FUNCTION Reader : INT
VAR
	numbers : ARRAY[1..5] OF INT := [12, 3, 6, 9];  // Your set of numbers
	
END_VAR

Random.number:=Random.number+3;
IF Random.number>12 THEN
	Random.number:=0;
END_IF

END_FUNCTION

(* stored: Version 1.1.0.1, ProductVersion 3.1.4024.12
   POU Reader: Id {9d2d486f-b22e-40c1-bfd5-bf17de1419d8}, SpecialFunc None *)
